FUNCTION WORD_TO_RANGE : REAL
VAR_INPUT
	X : WORD;
	low : REAL;
	high : REAL;
END_VAR


(*
version 1.1	10. mar. 2009
programmer 	hugo
tested by		tobias

Word_to_Range converts a Byte into a real between low and high.

*)

WORD_TO_RANGE := (high - low) * WORD_TO_REAL(X) * 0.00001525902189669640 + low;


(* revision history
hm	9. jan 2008	rev 1.0
	original version

hm	10. mar. 2009	rev 1.1
	improved code
*)

END_FUNCTION

(* stored: Version 1.1.0.1, ProductVersion 3.1.4022.7
   POU WORD_TO_RANGE: Id {499ba64f-2cf8-4425-9b97-8c31ae688f90}, SpecialFunc None *)
